// TIA Portal V20 export
TYPE "typeCmControlNodeInterlock"
// stored: Namespace Unit1.Em5
   STRUCT
      transferPnPLeftAxisX : "LER_typeAxisInterlock";
      transferPnPLeftAxisY : "LER_typeAxisInterlock";
      transferPnPLeftAxisZ : "LER_typeAxisInterlock";
      transferPnPRightAxisX : "LER_typeAxisInterlock";
      transferPnPRightAxisY : "LER_typeAxisInterlock";
      transferPnPRightAxisZ : "LER_typeAxisInterlock";
      transferPnPLeftClamp : "LER_typeTwoWayActuatorInterlock";
      transferPnPRightClamp : "LER_typeTwoWayActuatorInterlock";
   END_STRUCT;
END_TYPE
